(* PLC project waste-water, Generated TextualNotationConverter 1.0 *)
(* stored: creationDateTime 2025-07-30T12:00:00, modificationDateTime 2025-01-30T12:00:00 *)

FUNCTION_BLOCK ANALOG_IN
  VAR_INPUT
    Name : STRING;
    Description : STRING;
    Raw_Signal : REAL;
    PV_High : REAL;
    PV_Low : REAL;
    Scaling_Slope : REAL;
    Scaling_Offset : REAL;
    Alarm_Enable : BOOL;
  END_VAR
  VAR_OUTPUT
    PV : REAL;
    High_Alarm : BOOL;
    Low_Alarm : BOOL;
    General_Fault : BOOL;
  END_VAR

            
          
END_FUNCTION_BLOCK

FUNCTION_BLOCK BOOL_IN
  VAR_INPUT
    Name : STRING;
    Description : STRING;
    Bool_In : BOOL;
    Alarm_OnTrue : BOOL;
    Alarm_OnFalse : BOOL;
    Latch_Enable : BOOL;
    Reset_Latch : BOOL;
  END_VAR
  VAR_OUTPUT
    Bool_Out : BOOL;
    Alarm_Active : BOOL;
    Latched_Status : BOOL;
  END_VAR

            
          
END_FUNCTION_BLOCK

FUNCTION_BLOCK MOTOR_ON_OFF
  VAR_INPUT
    Name : STRING;
    Description : STRING;
    Start_Cmd : BOOL;
    Stop_Cmd : BOOL;
    Start_Delay : STRING;
    MinRunTime : STRING;
    Inhibit : BOOL;
  END_VAR
  VAR_OUTPUT
    Motor_Start_Out : BOOL;
    FB_Running : BOOL;
    FB_Trip : BOOL;
    Alarm_Start_Fail : BOOL;
    Alarm_Stop_Fail : BOOL;
  END_VAR

            
          
END_FUNCTION_BLOCK

FUNCTION_BLOCK MOTOR_VSD
  VAR_INPUT
    Name : STRING;
    Description : STRING;
    Start_Cmd : BOOL;
    Stop_Cmd : BOOL;
    Speed_SP : REAL;
    Accel_Ramp : STRING;
    Decel_Ramp : STRING;
    Inhibit : BOOL;
  END_VAR
  VAR_OUTPUT
    Speed_Out : REAL;
    FB_Running : BOOL;
    FB_Fault : BOOL;
    FB_Ready : BOOL;
    FB_ActualSpeed : REAL;
    Alarm_Speed_Deviation : BOOL;
    Alarm_Comm_Fail : BOOL;
  END_VAR

            
          
END_FUNCTION_BLOCK

FUNCTION_BLOCK PID_BASIC
  VAR_INPUT
    Name : STRING;
    Description : STRING;
    AUTO : BOOL;
    PV : REAL;
    SP : REAL;
    MV_MIN : REAL;
    MV_MAX : REAL;
    X0 : REAL;
    KP : REAL;
    TR : REAL;
    TD : REAL;
    PV_High : REAL;
    PV_Low : REAL;
    Deviation_Limit : REAL;
    Inhibit : BOOL;
  END_VAR
  VAR_OUTPUT
    PV_High_Alarm : BOOL;
    PV_Low_Alarm : BOOL;
    Deviation_Alarm : BOOL;
    XOUT : REAL;
  END_VAR

            
          
END_FUNCTION_BLOCK

FUNCTION_BLOCK VALVE_ON_OFF
  VAR_INPUT
    Name : STRING;
    Description : STRING;
    Open_Cmd : BOOL;
    Close_Cmd : BOOL;
    Timeout : STRING;
    Inhibit : BOOL;
  END_VAR
  VAR_OUTPUT
    FB_Opened : BOOL;
    FB_Closed : BOOL;
    Valve_Open_Out : BOOL;
    Valve_Close_Out : BOOL;
    Alarm_Position_Error : BOOL;
    Alarm_General : BOOL;
  END_VAR

            
          
END_FUNCTION_BLOCK

PROGRAM Sec2
  VAR
    LS_101_WetWellLevel_PV_m : REAL;
    FT_101_InfluentFlow_PV_m3ph : REAL;
    PIC_101_WetWellLevel_MV_Pct : REAL;
    P_101A_Speed_Command_Pct : REAL;
    P_101B_Speed_Command_Pct : REAL;
    P101_LevelTrips_Active : BOOL;
    VG101_Inhibit_Active : BOOL;
    BS101_Disable_Active : BOOL;
    P_101A_Start_Cmd : BOOL;
    P_101B_Start_Cmd : BOOL;
  END_VAR
  VAR
    FT-101 : ANALOG_IN;
    LS-101 : ANALOG_IN;
    PIC-101 : PID_BASIC;
    P-101A : MOTOR_VSD;
    P-101B : MOTOR_VSD;
    XV-101 : VALVE_ON_OFF;
    BS-101 : BOOL_IN;
    VG-101 : MOTOR_ON_OFF;
  END_VAR
  VAR  (* added by the conversion: wires and edge detectors of the diagram *)
    _OR3_OUT : BOOL;
    _OR1_OUT : BOOL;
    _AND6_OUT : BOOL;
    _AND11_OUT : BOOL;
    _OR2_OUT : BOOL;
    _GT4_OUT : BOOL;
  END_VAR

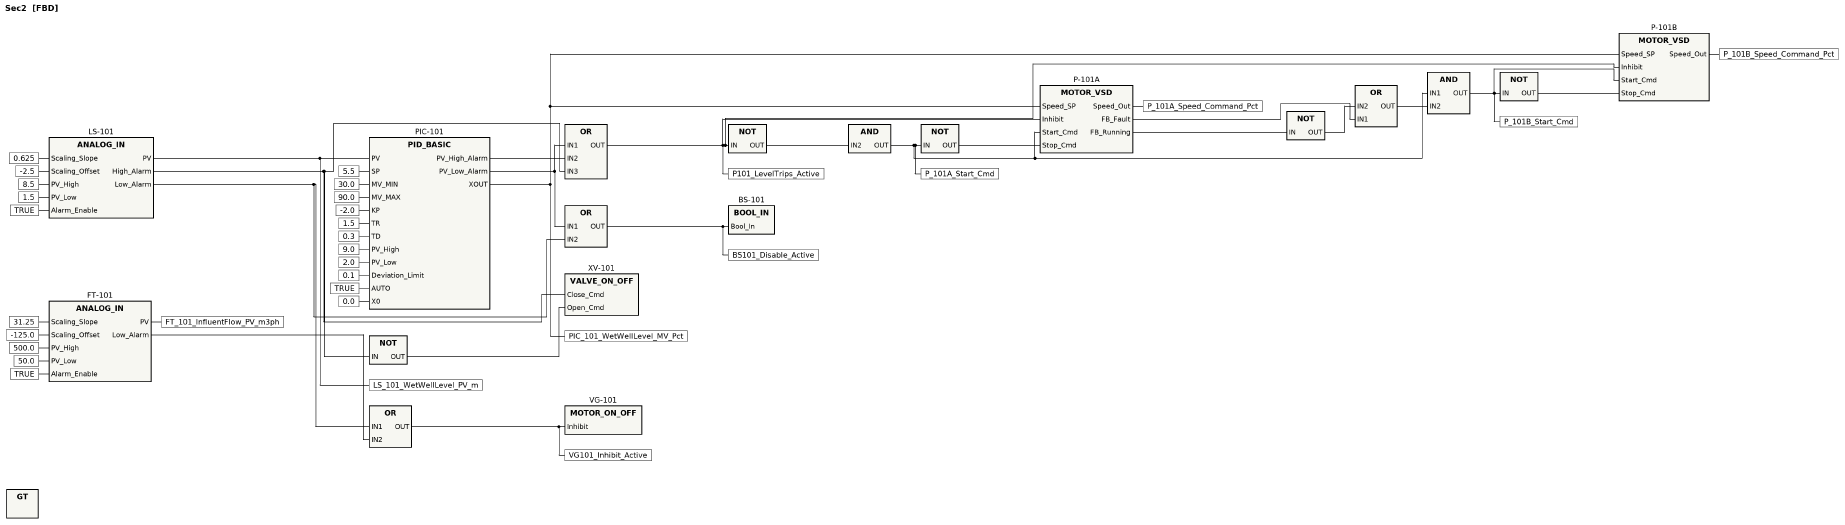
(* FBD diagram, written out as Structured Text *)
LS-101(Scaling_Slope := 0.625, Scaling_Offset := -2.5, PV_High := 8.5, PV_Low := 1.5, Alarm_Enable := TRUE);
PIC-101(PV := LS-101.PV, SP := 5.5, MV_MIN := 30.0, MV_MAX := 90.0, KP := -2.0, TR := 1.5, TD := 0.3, PV_High := 9.0, PV_Low := 2.0, Deviation_Limit := 0.1, AUTO := TRUE, X0 := 0.0);
_OR3_OUT := PIC-101.PV_Low_Alarm OR LS-101.Low_Alarm;
BS101_Disable_Active := _OR3_OUT;
FT-101(Scaling_Slope := 31.25, Scaling_Offset := -125.0, PV_High := 500.0, PV_Low := 50.0, Alarm_Enable := TRUE);
FT_101_InfluentFlow_PV_m3ph := FT-101.PV;
LS_101_WetWellLevel_PV_m := LS-101.PV;
_OR1_OUT := PIC-101.PV_Low_Alarm OR PIC-101.PV_High_Alarm OR LS-101.High_Alarm;
P101_LevelTrips_Active := _OR1_OUT;
PIC_101_WetWellLevel_MV_Pct := PIC-101.XOUT;
_AND6_OUT := AND(NOT _OR1_OUT);
P-101A(Speed_SP := PIC-101.XOUT, Inhibit := _OR1_OUT, Start_Cmd := _AND6_OUT, Stop_Cmd := NOT _AND6_OUT);
P_101A_Speed_Command_Pct := P-101A.Speed_Out;
P_101A_Start_Cmd := _AND6_OUT;
_AND11_OUT := _AND6_OUT AND (NOT P-101A.FB_Running OR P-101A.FB_Fault);
P-101B(Speed_SP := PIC-101.XOUT, Inhibit := _OR1_OUT, Start_Cmd := _AND11_OUT, Stop_Cmd := NOT _AND11_OUT);
P_101B_Speed_Command_Pct := P-101B.Speed_Out;
P_101B_Start_Cmd := _AND11_OUT;
_OR2_OUT := LS-101.Low_Alarm OR FT-101.Low_Alarm;
VG101_Inhibit_Active := _OR2_OUT;
_GT4_OUT := GT();
XV-101(Close_Cmd := LS-101.High_Alarm, Open_Cmd := NOT LS-101.High_Alarm);
BS-101(Bool_In := _OR3_OUT);
VG-101(Inhibit := _OR2_OUT);
END_PROGRAM

FUNCTION_BLOCK DIGITAL_IN
  VAR_INPUT
    Name : STRING;
    Description : STRING;
    DI_Raw : BOOL;
    DebounceTime : STRING;
    EnableAlarm : BOOL;
  END_VAR
  VAR_OUTPUT
    DI_Out : BOOL;
    Fault_State : BOOL;
  END_VAR

            
          
END_FUNCTION_BLOCK

FUNCTION_BLOCK DUTY_STANDBY
  VAR_INPUT
    Name : STRING;
    Description : STRING;
    Enable : BOOL;
    StartRequest : BOOL;
    AlternateEnable : BOOL;
    ForcePumpA : BOOL;
    ForcePumpB : BOOL;
    DutyElapsed : BOOL;
    MinRunElapsed : BOOL;
    SwitchoverDelayElapsed : BOOL;
    StartTimeoutElapsed : BOOL;
    PumpA_RunFB : BOOL;
    PumpB_RunFB : BOOL;
    PumpA_Fault : BOOL;
    PumpB_Fault : BOOL;
    Reset : BOOL;
    Inhibit : BOOL;
  END_VAR
  VAR_OUTPUT
    CmdPumpA : BOOL;
    CmdPumpB : BOOL;
    ActiveIsA : BOOL;
    SwitchedDueToDuty : BOOL;
    SwitchedDueToFailure : BOOL;
    Alarm_FailedStart_A : BOOL;
    Alarm_FailedStart_B : BOOL;
    Alarm_NoAvailablePump : BOOL;
  END_VAR

            
          
END_FUNCTION_BLOCK

FUNCTION_BLOCK MOTOR_2SPD
  VAR_INPUT
    Name : STRING;
    Description : STRING;
    Start_Cmd : BOOL;
    Stop_Cmd : BOOL;
    Speed_High_Cmd : BOOL;
    Speed_Low_Cmd : BOOL;
    Inhibit : BOOL;
  END_VAR
  VAR_OUTPUT
    Motor_Start_Out : BOOL;
    FB_Running : BOOL;
    FB_Trip : BOOL;
    FB_HighSpeed : BOOL;
    FB_LowSpeed : BOOL;
    Alarm_Speed_Error : BOOL;
  END_VAR

            
          
END_FUNCTION_BLOCK

FUNCTION_BLOCK RATIO_CONTROL
  VAR_INPUT
    Name : STRING;
    Description : STRING;
    Auto : BOOL;
    PrimaryPV : REAL;
    SecondaryPV : REAL;
    RatioSP : REAL;
    Bias : REAL;
    TrimKp : REAL;
    TrimTi : STRING;
    MV_MIN : REAL;
    MV_MAX : REAL;
    ManOut : REAL;
    Inhibit : BOOL;
  END_VAR
  VAR_OUTPUT
    SlaveSP : REAL;
    ActiveRatio : REAL;
    RatioErr : REAL;
  END_VAR

            
          
END_FUNCTION_BLOCK

FUNCTION_BLOCK SPLIT_RANGE
  VAR_INPUT
    Name : STRING;
    Description : STRING;
    IN : REAL;
    Split_Point : REAL;
    Output1_Start : REAL;
    Output1_End : REAL;
    Output2_Start : REAL;
    Output2_End : REAL;
  END_VAR
  VAR_OUTPUT
    OUT1 : REAL;
    OUT2 : REAL;
  END_VAR

            
          
END_FUNCTION_BLOCK

FUNCTION_BLOCK VALVE_ELECTRIC
  VAR_INPUT
    Name : STRING;
    Description : STRING;
    Control_Signal : REAL;
    Manual_Mode : BOOL;
    Manual_Position : REAL;
    Open_Limit : REAL;
    Close_Limit : REAL;
    Timeout : STRING;
    Inhibit : BOOL;
  END_VAR
  VAR_OUTPUT
    Valve_Position : REAL;
    Feedback_Pos : REAL;
    Valve_Moving : BOOL;
    Position_Error : BOOL;
    Alarm : BOOL;
  END_VAR

            
          
END_FUNCTION_BLOCK

FUNCTION_BLOCK VOTING_ANALOG
  VAR_INPUT
    Name : STRING;
    Description : STRING;
    Input1 : REAL;
    Input2 : REAL;
    Input3 : REAL;
    Deviation_Limit : REAL;
    Voting_Scheme : STRING;
    EnableAlarm : BOOL;
    Inhibit : BOOL;
  END_VAR
  VAR_OUTPUT
    Voted_Output : REAL;
    Sensor1_Fault : BOOL;
    Sensor2_Fault : BOOL;
    Sensor3_Fault : BOOL;
    Alarm_Voting_Error : BOOL;
    Healthy_Sensors_Count : INT;
  END_VAR

            
          
END_FUNCTION_BLOCK

PROGRAM Sec4
  VAR
    FT301_InfluentFlow_PV : REAL;
    FT302_SludgeFlow_PV : REAL;
    LS301_WeirLevel_PV : REAL;
    PS301_SludgePressure_PV : REAL;
    FT302_SludgeFlow_SP : REAL;
  END_VAR
  VAR
    FT-301 : ANALOG_IN;
    FT-302 : ANALOG_IN;
    LS-301 : ANALOG_IN;
    PS-301 : ANALOG_IN;
    SS-301 : DIGITAL_IN;
    FV-102 : VALVE_ELECTRIC;
    FFIC-303 : RATIO_CONTROL;
    FIC-302 : PID_BASIC;
  END_VAR
  VAR  (* added by the conversion: wires and edge detectors of the diagram *)
    _GT52_OUT : BOOL;
    _OR53_OUT : BOOL;
  END_VAR

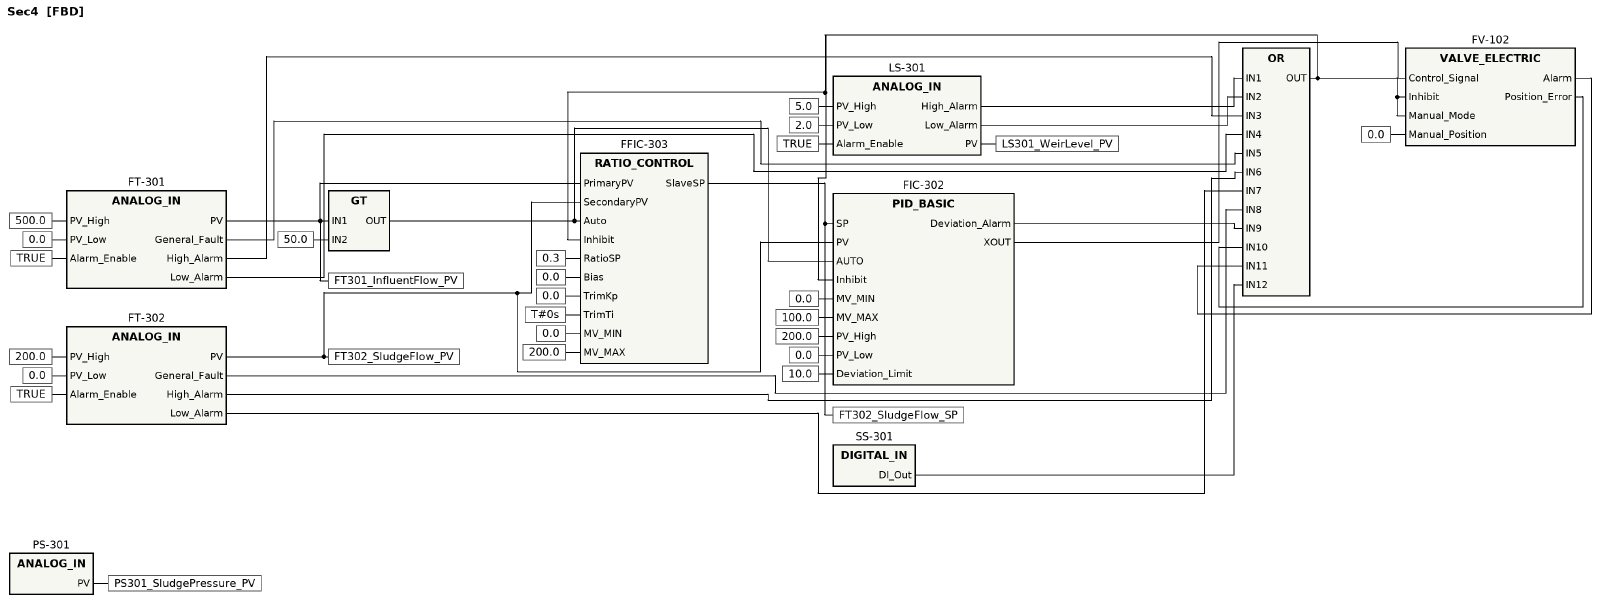
(* FBD diagram, written out as Structured Text *)
FT-301(PV_High := 500.0, PV_Low := 0.0, Alarm_Enable := TRUE);
FT301_InfluentFlow_PV := FT-301.PV;
FT-302(PV_High := 200.0, PV_Low := 0.0, Alarm_Enable := TRUE);
FT302_SludgeFlow_PV := FT-302.PV;
_GT52_OUT := FT-301.PV > 50.0;
LS-301(PV_High := 5.0, PV_Low := 2.0, Alarm_Enable := TRUE);
FIC-302(SP := FFIC-303.SlaveSP, PV := FT-302.PV, AUTO := _GT52_OUT, Inhibit := _OR53_OUT, MV_MIN := 0.0, MV_MAX := 100.0, PV_High := 200.0, PV_Low := 0.0, Deviation_Limit := 10.0);
FV-102(Control_Signal := FIC-302.XOUT, Inhibit := _OR53_OUT, Manual_Mode := _OR53_OUT, Manual_Position := 0.0);
SS-301();
_OR53_OUT := LS-301.High_Alarm OR LS-301.Low_Alarm OR FT-301.High_Alarm OR FT-301.Low_Alarm OR FT-301.General_Fault OR FT-302.High_Alarm OR FT-302.Low_Alarm OR FT-302.General_Fault OR FIC-302.Deviation_Alarm OR FV-102.Position_Error OR FV-102.Alarm OR SS-301.DI_Out;
FFIC-303(PrimaryPV := FT-301.PV, SecondaryPV := FT-302.PV, Auto := _GT52_OUT, Inhibit := _OR53_OUT, RatioSP := 0.3, Bias := 0.0, TrimKp := 0.0, TrimTi := T#0s, MV_MIN := 0.0, MV_MAX := 200.0);
FT302_SludgeFlow_SP := FFIC-303.SlaveSP;
LS301_WeirLevel_PV := LS-301.PV;
PS-301();
PS301_SludgePressure_PV := PS-301.PV;
END_PROGRAM

PROGRAM Sec7
  VAR
    PT-601A_DischargePressure_PV : REAL;
    PT-601B_DischargePressure_PV : REAL;
    CL-601_ActiveIsA : BOOL;
    PS-601_ActiveIsA : BOOL;
  END_VAR
  VAR
    CL-601A : MOTOR_ON_OFF;
    CL-601B : MOTOR_ON_OFF;
    PS-601A : MOTOR_ON_OFF;
    PS-601B : MOTOR_ON_OFF;
    PT-601A : ANALOG_IN;
    PT-601B : ANALOG_IN;
    LS-601 : DIGITAL_IN;
    VS-601A : VALVE_ELECTRIC;
    VS-601B : VALVE_ELECTRIC;
    CL-601A_CL-601B : DUTY_STANDBY;
    PS-601A_PS-601B : DUTY_STANDBY;
    Clar_MinRunTimer_TON : TON;
    Clar_DutyTimer_TON : TON;
    Clar_SwitchoverDelay_TON : TON;
    Pump_MinRunTimer_TON : TON;
    Pump_DutyTimer_TON : TON;
    Pump_SwitchoverDelay_TON : TON;
  END_VAR
  VAR  (* added by the conversion: wires and edge detectors of the diagram *)
    _OR89_OUT : BOOL;
    _OR91_OUT : BOOL;
  END_VAR

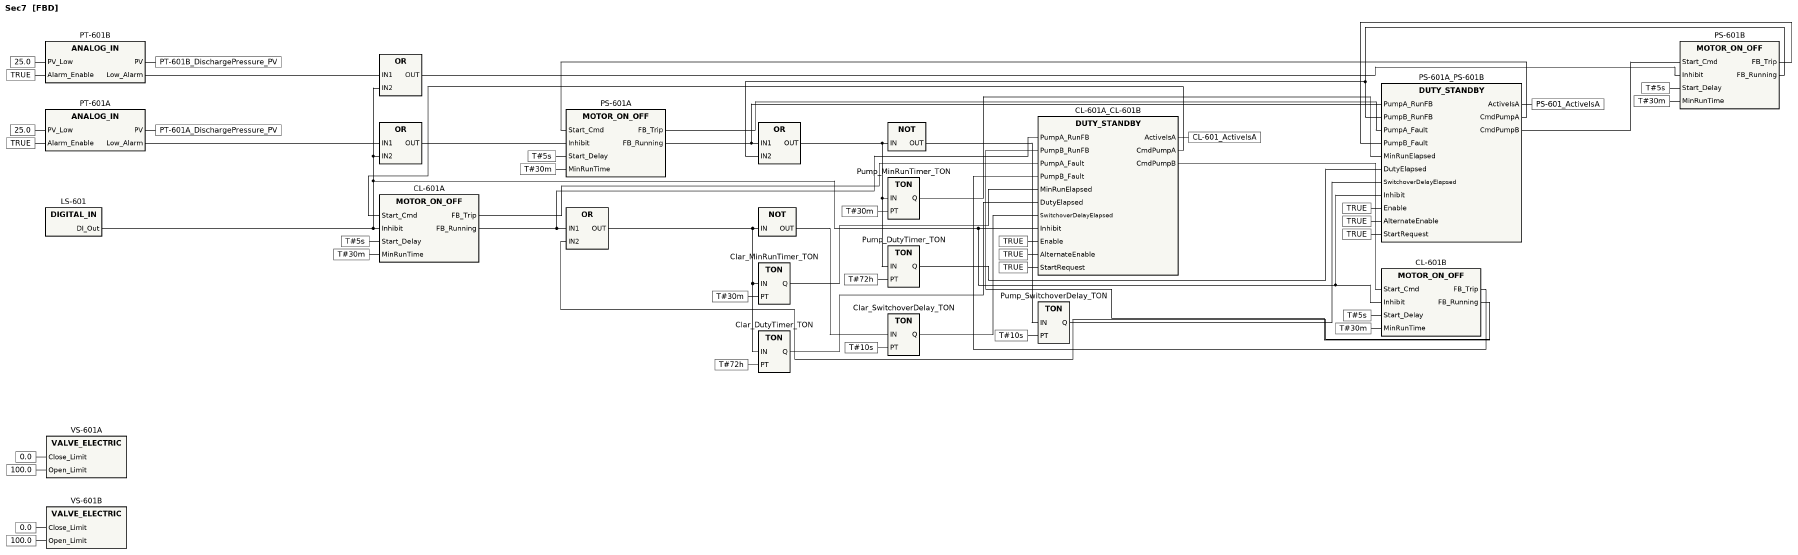
(* FBD diagram, written out as Structured Text *)
LS-601();
CL-601A(Start_Cmd := CL-601A_CL-601B.CmdPumpA, Inhibit := LS-601.DI_Out, Start_Delay := T#5s, MinRunTime := T#30m);
CL-601B(Start_Cmd := CL-601A_CL-601B.CmdPumpB, Inhibit := LS-601.DI_Out, Start_Delay := T#5s, MinRunTime := T#30m);
_OR89_OUT := CL-601A.FB_Running OR CL-601B.FB_Running;
Clar_MinRunTimer_TON(IN := _OR89_OUT, PT := T#30m);
Clar_DutyTimer_TON(IN := _OR89_OUT, PT := T#72h);
Clar_SwitchoverDelay_TON(IN := NOT _OR89_OUT, PT := T#10s);
CL-601A_CL-601B(PumpA_RunFB := CL-601A.FB_Running, PumpB_RunFB := CL-601B.FB_Running, PumpA_Fault := CL-601A.FB_Trip, PumpB_Fault := CL-601B.FB_Trip, MinRunElapsed := Clar_MinRunTimer_TON.Q, DutyElapsed := Clar_DutyTimer_TON.Q, SwitchoverDelayElapsed := Clar_SwitchoverDelay_TON.Q, Inhibit := LS-601.DI_Out, Enable := TRUE, AlternateEnable := TRUE, StartRequest := TRUE);
CL-601_ActiveIsA := CL-601A_CL-601B.ActiveIsA;
PT-601A(PV_Low := 25.0, Alarm_Enable := TRUE);
PS-601A(Start_Cmd := PS-601A_PS-601B.CmdPumpA, Inhibit := PT-601A.Low_Alarm OR LS-601.DI_Out, Start_Delay := T#5s, MinRunTime := T#30m);
PT-601B(PV_Low := 25.0, Alarm_Enable := TRUE);
PS-601B(Start_Cmd := PS-601A_PS-601B.CmdPumpB, Inhibit := PT-601B.Low_Alarm OR LS-601.DI_Out, Start_Delay := T#5s, MinRunTime := T#30m);
_OR91_OUT := PS-601A.FB_Running OR PS-601B.FB_Running;
Pump_MinRunTimer_TON(IN := _OR91_OUT, PT := T#30m);
Pump_DutyTimer_TON(IN := _OR91_OUT, PT := T#72h);
Pump_SwitchoverDelay_TON(IN := NOT _OR91_OUT, PT := T#10s);
PS-601A_PS-601B(PumpA_RunFB := PS-601A.FB_Running, PumpB_RunFB := PS-601B.FB_Running, PumpA_Fault := PS-601A.FB_Trip, PumpB_Fault := PS-601B.FB_Trip, MinRunElapsed := Pump_MinRunTimer_TON.Q, DutyElapsed := Pump_DutyTimer_TON.Q, SwitchoverDelayElapsed := Pump_SwitchoverDelay_TON.Q, Inhibit := LS-601.DI_Out, Enable := TRUE, AlternateEnable := TRUE, StartRequest := TRUE);
PS-601_ActiveIsA := PS-601A_PS-601B.ActiveIsA;
PT-601A_DischargePressure_PV := PT-601A.PV;
PT-601B_DischargePressure_PV := PT-601B.PV;
VS-601A(Close_Limit := 0.0, Open_Limit := 100.0);
VS-601B(Close_Limit := 0.0, Open_Limit := 100.0);
END_PROGRAM

PROGRAM Sec9
  VAR
    FT_801_EffluentFlow_PV : REAL;
    CL_801_ChlorineFlow_SP : REAL;
    DC_801_DechlorFlow_SP : REAL;
    XV_106_FullyOpen_FB : BOOL;
    CL_801_Running_FB : BOOL;
    DC_801_Running_FB : BOOL;
  END_VAR
  VAR
    FT-801 : ANALOG_IN;
    FIC-101 : RATIO_CONTROL;
    FIC-102 : RATIO_CONTROL;
    CL-801 : MOTOR_VSD;
    DC-801 : MOTOR_VSD;
    LV-105 : VALVE_ELECTRIC;
    XV-106 : VALVE_ON_OFF;
    UV-801 : MOTOR_ON_OFF;
  END_VAR
  VAR  (* added by the conversion: wires and edge detectors of the diagram *)
    _OR151_OUT : BOOL;
    _OR159_OUT : BOOL;
    _NOT149_OUT : BOOL;
  END_VAR

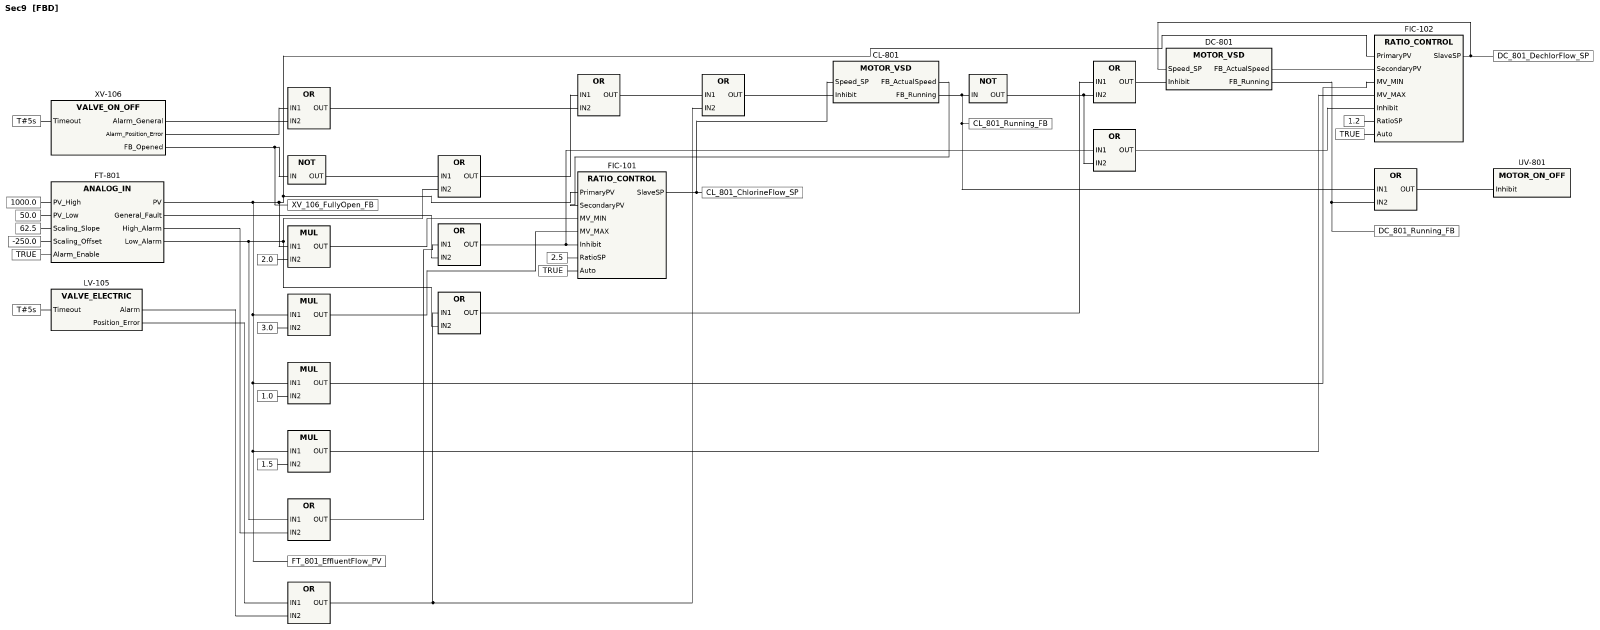
(* FBD diagram, written out as Structured Text *)
FT-801(PV_High := 1000.0, PV_Low := 50.0, Scaling_Slope := 62.5, Scaling_Offset := -250.0, Alarm_Enable := TRUE);
XV-106(Timeout := T#5s);
LV-105(Timeout := T#5s);
_OR151_OUT := LV-105.Position_Error OR LV-105.Alarm;
CL-801(Speed_SP := FIC-101.SlaveSP, Inhibit := NOT XV-106.FB_Opened OR FT-801.Low_Alarm OR XV-106.Alarm_Position_Error OR XV-106.Alarm_General OR _OR151_OUT);
_OR159_OUT := FT-801.Low_Alarm OR FT-801.High_Alarm OR FT-801.General_Fault;
FIC-101(PrimaryPV := FT-801.PV, SecondaryPV := CL-801.FB_ActualSpeed, MV_MIN := FT-801.PV * 2.0, MV_MAX := FT-801.PV * 3.0, Inhibit := _OR159_OUT, RatioSP := 2.5, Auto := TRUE);
CL_801_ChlorineFlow_SP := FIC-101.SlaveSP;
CL_801_Running_FB := CL-801.FB_Running;
_NOT149_OUT := NOT CL-801.FB_Running;
DC-801(Speed_SP := FIC-102.SlaveSP, Inhibit := _OR151_OUT OR FT-801.Low_Alarm OR _NOT149_OUT);
FIC-102(PrimaryPV := FT-801.PV, SecondaryPV := DC-801.FB_ActualSpeed, MV_MIN := FT-801.PV * 1.0, MV_MAX := FT-801.PV * 1.5, Inhibit := _OR159_OUT OR _NOT149_OUT, RatioSP := 1.2, Auto := TRUE);
DC_801_DechlorFlow_SP := FIC-102.SlaveSP;
DC_801_Running_FB := DC-801.FB_Running;
FT_801_EffluentFlow_PV := FT-801.PV;
XV_106_FullyOpen_FB := XV-106.FB_Opened;
UV-801(Inhibit := CL-801.FB_Running OR DC-801.FB_Running);
END_PROGRAM

PROGRAM Sec10
  VAR
    FT_901_FlowRate : REAL;
    LS_901_LevelPercent : REAL;
    P_901A_Running : BOOL;
    P_901B_Running : BOOL;
    P_901AB_DutyActiveIsA : BOOL;
    P_901AB_SwitchedDueToDuty : BOOL;
    P_901AB_SwitchedDueToFailure : BOOL;
  END_VAR
  VAR
    FT-901 : ANALOG_IN;
    LS-901 : ANALOG_IN;
    P-901A : MOTOR_ON_OFF;
    P-901B : MOTOR_ON_OFF;
    XV-102 : VALVE_ON_OFF;
    P-901AB : DUTY_STANDBY;
  END_VAR
  VAR  (* added by the conversion: wires and edge detectors of the diagram *)
    _GT194_OUT : BOOL;
    _GT197_OUT : BOOL;
    _TON199_OUT : BOOL;
    _TON201_OUT : BOOL;
    _OR190_OUT : BOOL;
  END_VAR

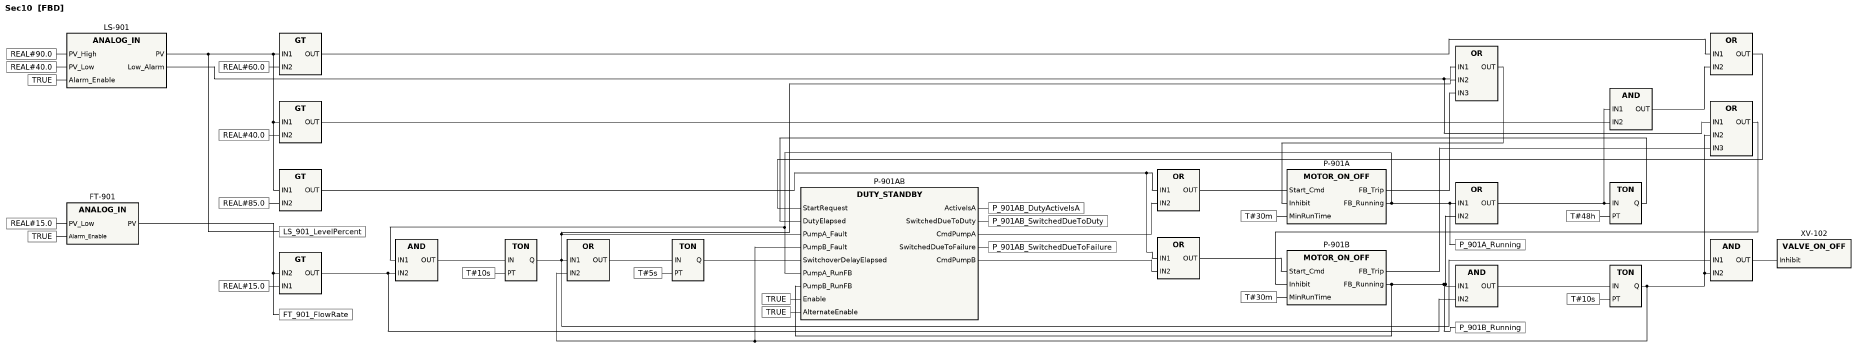
(* FBD diagram, written out as Structured Text *)
FT-901(PV_Low := REAL#15.0, Alarm_Enable := TRUE);
FT_901_FlowRate := FT-901.PV;
LS-901(PV_High := REAL#90.0, PV_Low := REAL#40.0, Alarm_Enable := TRUE);
LS_901_LevelPercent := LS-901.PV;
_GT194_OUT := LS-901.PV > REAL#85.0;
_GT197_OUT := FT-901.PV > REAL#15.0;
_TON199_OUT := TON(P-901A.FB_Running AND _GT197_OUT, T#10s);
P-901A(Start_Cmd := _GT194_OUT OR P-901AB.CmdPumpA, Inhibit := LS-901.Low_Alarm OR _TON199_OUT OR P-901A.FB_Trip, MinRunTime := T#30m);
_TON201_OUT := TON(P-901B.FB_Running AND _GT197_OUT, T#10s);
P-901B(Start_Cmd := _GT194_OUT OR P-901AB.CmdPumpB, Inhibit := LS-901.Low_Alarm OR _TON201_OUT OR P-901B.FB_Trip, MinRunTime := T#30m);
_OR190_OUT := P-901A.FB_Running OR P-901B.FB_Running;
P-901AB(StartRequest := LS-901.PV > REAL#60.0 OR _OR190_OUT AND LS-901.PV > REAL#40.0, DutyElapsed := TON(_OR190_OUT, T#48h), PumpA_Fault := _TON199_OUT, PumpB_Fault := _TON201_OUT, SwitchoverDelayElapsed := TON(_TON199_OUT OR _TON201_OUT, T#5s), PumpA_RunFB := P-901A.FB_Running, PumpB_RunFB := P-901B.FB_Running, Enable := TRUE, AlternateEnable := TRUE);
P_901AB_DutyActiveIsA := P-901AB.ActiveIsA;
P_901AB_SwitchedDueToDuty := P-901AB.SwitchedDueToDuty;
P_901AB_SwitchedDueToFailure := P-901AB.SwitchedDueToFailure;
P_901A_Running := P-901A.FB_Running;
P_901B_Running := P-901B.FB_Running;
XV-102(Inhibit := _TON199_OUT AND _TON201_OUT);
END_PROGRAM

PROGRAM Sec11
  VAR
    FIT_104_InfluentFlow_PV : REAL;
    FIC_106_SP_From_FFIC_107 : REAL;
  END_VAR
  VAR
    FIT-104 : ANALOG_IN;
    FFIC-107 : RATIO_CONTROL;
    FIC-106 : PID_BASIC;
    CD-1001 : MOTOR_VSD;
    PV-101 : VALVE_ELECTRIC;
    XV-102 : VALVE_ON_OFF;
  END_VAR

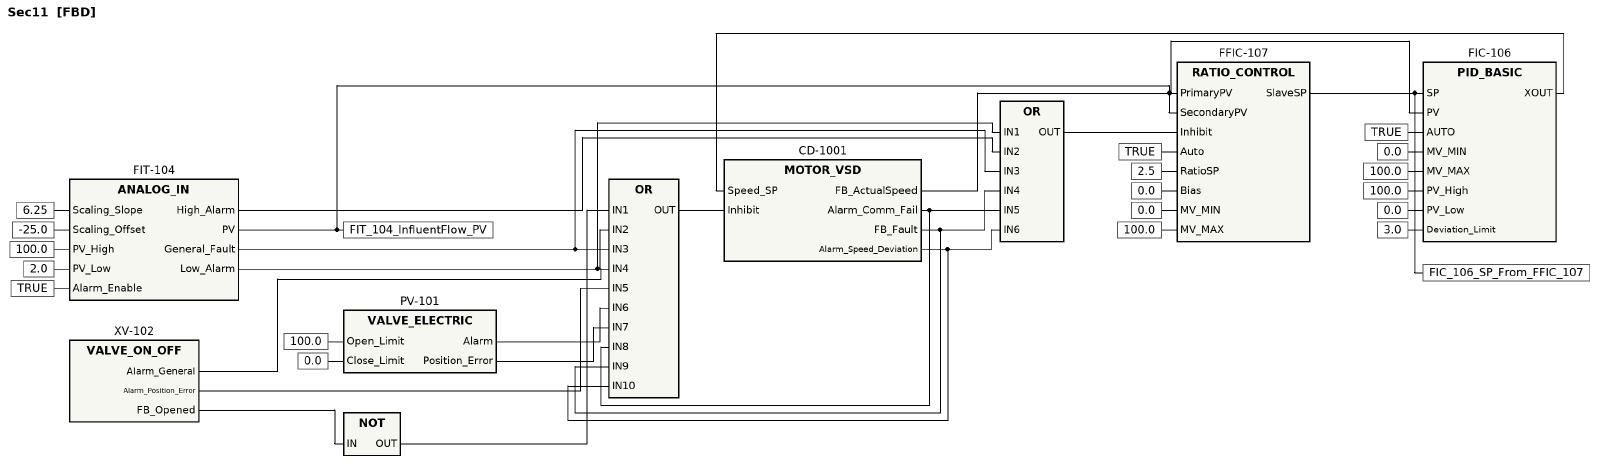
(* FBD diagram, written out as Structured Text *)
FIT-104(Scaling_Slope := 6.25, Scaling_Offset := -25.0, PV_High := 100.0, PV_Low := 2.0, Alarm_Enable := TRUE);
FIC-106(SP := FFIC-107.SlaveSP, PV := CD-1001.FB_ActualSpeed, AUTO := TRUE, MV_MIN := 0.0, MV_MAX := 100.0, PV_High := 100.0, PV_Low := 0.0, Deviation_Limit := 3.0);
XV-102();
PV-101(Open_Limit := 100.0, Close_Limit := 0.0);
CD-1001(Speed_SP := FIC-106.XOUT, Inhibit := NOT XV-102.FB_Opened OR FIT-104.Low_Alarm OR FIT-104.General_Fault OR XV-102.Alarm_General OR XV-102.Alarm_Position_Error OR PV-101.Alarm OR PV-101.Position_Error OR CD-1001.Alarm_Comm_Fail OR CD-1001.FB_Fault OR CD-1001.Alarm_Speed_Deviation);
FFIC-107(PrimaryPV := FIT-104.PV, SecondaryPV := CD-1001.FB_ActualSpeed, Inhibit := FIT-104.Low_Alarm OR FIT-104.High_Alarm OR FIT-104.General_Fault OR CD-1001.FB_Fault OR CD-1001.Alarm_Comm_Fail OR CD-1001.Alarm_Speed_Deviation, Auto := TRUE, RatioSP := 2.5, Bias := 0.0, MV_MIN := 0.0, MV_MAX := 100.0);
FIC_106_SP_From_FFIC_107 := FFIC-107.SlaveSP;
FIT_104_InfluentFlow_PV := FIT-104.PV;
END_PROGRAM

PROGRAM Sec12
  VAR
    IIC101_Raw_mA : REAL;
    LV104_Raw_mA : REAL;
    IIC101_Solids_PV : REAL;
    IIC103_MV_to_PV102 : REAL;
    LV104_Level_PV : REAL;
  END_VAR
  VAR
    IIC-101 : ANALOG_IN;
    LV-104 : ANALOG_IN;
    IIC-103 : PID_BASIC;
    IIC-105 : BOOL_IN;
    PV-102 : VALVE_ELECTRIC;
    OC-1101 : VALVE_ON_OFF;
  END_VAR

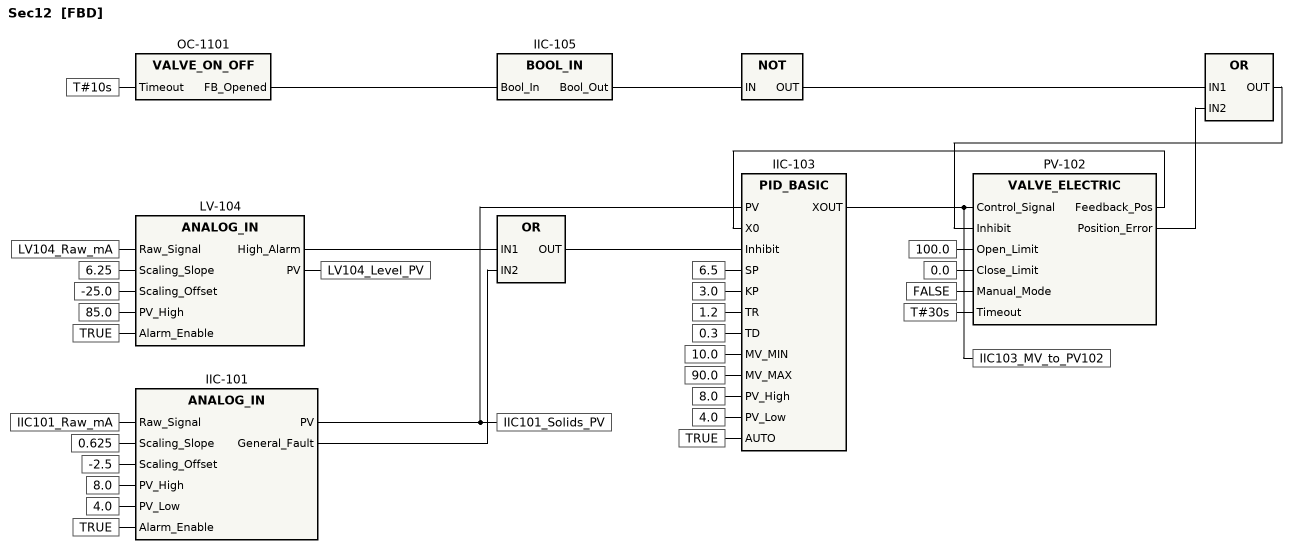
(* FBD diagram, written out as Structured Text *)
IIC-101(Raw_Signal := IIC101_Raw_mA, Scaling_Slope := 0.625, Scaling_Offset := -2.5, PV_High := 8.0, PV_Low := 4.0, Alarm_Enable := TRUE);
IIC101_Solids_PV := IIC-101.PV;
OC-1101(Timeout := T#10s);
IIC-105(Bool_In := OC-1101.FB_Opened);
PV-102(Control_Signal := IIC-103.XOUT, Inhibit := NOT IIC-105.Bool_Out OR PV-102.Position_Error, Open_Limit := 100.0, Close_Limit := 0.0, Manual_Mode := FALSE, Timeout := T#30s);
LV-104(Raw_Signal := LV104_Raw_mA, Scaling_Slope := 6.25, Scaling_Offset := -25.0, PV_High := 85.0, Alarm_Enable := TRUE);
IIC-103(PV := IIC-101.PV, X0 := PV-102.Feedback_Pos, Inhibit := LV-104.High_Alarm OR IIC-101.General_Fault, SP := 6.5, KP := 3.0, TR := 1.2, TD := 0.3, MV_MIN := 10.0, MV_MAX := 90.0, PV_High := 8.0, PV_Low := 4.0, AUTO := TRUE);
IIC103_MV_to_PV102 := IIC-103.XOUT;
LV104_Level_PV := LV-104.PV;
END_PROGRAM

CONFIGURATION Config0
  RESOURCE Res0 ON PLC
    TASK task0(INTERVAL := T#20ms, PRIORITY := 0);
    PROGRAM instance0 WITH task0 : Sec2;
    PROGRAM instance_1 WITH task0 : Sec4;
    PROGRAM instance_2 WITH task0 : Sec7;
    PROGRAM instance_3 WITH task0 : Sec9;
    PROGRAM instance_4 WITH task0 : Sec10;
    PROGRAM instance_5 WITH task0 : Sec11;
    PROGRAM instance_6 WITH task0 : Sec12;
  END_RESOURCE
END_CONFIGURATION
